ABB RAPID module: Module1.mod

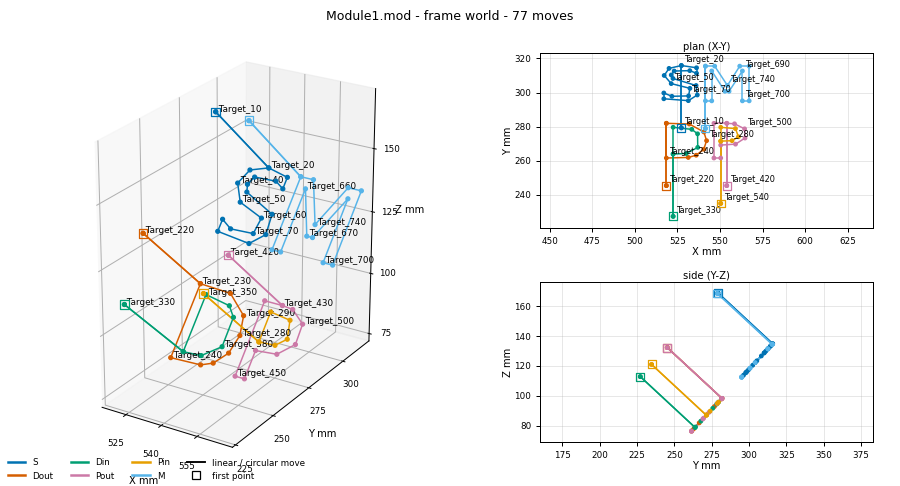
[picture p0: tool path of Module1.mod in frame world, 77 of 79 moves have a stored position in this frame; points joined in program order, loops and branches not executed]
MODULE Module1
        CONST robtarget Target_10:=[[155.704254378,97.181037963,47.999905215],[-0.000000229,0.899659187,0.436592885,-0.000000111],[0,0,-2,0],[9E+09,9E+09,9E+09,9E+09,9E+09,9E+09]];
    CONST robtarget Target_20:=[[155.704254378,97.181063465,-2.000094786],[-0.000000229,0.899659187,0.436592885,-0.000000111],[0,0,-2,0],[9E+09,9E+09,9E+09,9E+09,9E+09,9E+09]];
    CONST robtarget Target_30:=[[162.948986955,99.648648555,-2.000093527],[-0.000000246,0.899659158,0.436592946,0.000000066],[0,0,-2,0],[9E+09,9E+09,9E+09,9E+09,9E+09,9E+09]];
    CONST robtarget Target_40:=[[165.793395383,105.762911115,-2.000090408],[0.00000023,0.899659288,0.436592677,0.000000112],[0,0,-2,0],[9E+09,9E+09,9E+09,9E+09,9E+09,9E+09]];
    CONST robtarget Target_50:=[[161.67264984,112.800998636,-2.000086819],[0.00000023,0.899659288,0.436592677,0.000000111],[0,0,-2,0],[9E+09,9E+09,9E+09,9E+09,9E+09,9E+09]];
    CONST robtarget Target_60:=[[150.659683876,116.873121812,-2.000084742],[0.00000023,0.899659288,0.436592678,0.000000112],[0,0,-2,0],[9E+09,9E+09,9E+09,9E+09,9E+09,9E+09]];
    CONST robtarget Target_70:=[[151.461952919,123.42498567,-2.0000814],[-0.000000248,0.899659158,0.436592944,0.000000058],[0,0,-2,0],[9E+09,9E+09,9E+09,9E+09,9E+09,9E+09]];
    CONST robtarget Target_80:=[[161.259359726,123.777497824,-2.000081221],[-0.00000017,0.899659215,0.436592827,-0.00000019],[0,0,-2,0],[9E+09,9E+09,9E+09,9E+09,9E+09,9E+09]];
    CONST robtarget Target_90:=[[166.012196031,120.908778214,-2.000082684],[-0.000000229,0.899659187,0.436592885,-0.000000111],[0,0,-2,0],[9E+09,9E+09,9E+09,9E+09,9E+09,9E+09]];
    CONST robtarget Target_100:=[[166.012196031,125.916881941,-2.000080129],[0.00000023,0.899659288,0.436592677,0.000000112],[0,0,-2,0],[9E+09,9E+09,9E+09,9E+09,9E+09,9E+09]];
    CONST robtarget Target_110:=[[151.595664427,127.545731212,-2.000079299],[0.00000023,0.899659288,0.436592678,0.000000112],[0,0,-2,0],[9E+09,9E+09,9E+09,9E+09,9E+09,9E+09]];
    CONST robtarget Target_120:=[[146.332293276,122.634872217,-2.000081803],[0.000000229,0.899659287,0.436592678,0.000000111],[0,0,-2,0],[9E+09,9E+09,9E+09,9E+09,9E+09,9E+09]];
    CONST robtarget Target_130:=[[147.049473179,114.454159089,-2.000085976],[-0.000000049,0.899659258,0.436592738,-0.00000025],[0,0,-2,0],[9E+09,9E+09,9E+09,9E+09,9E+09,9E+09]];
    CONST robtarget Target_140:=[[160.627268965,108.376363303,-2.000089076],[-0.00000007,0.899659251,0.436592752,-0.000000245],[0,0,-2,0],[9E+09,9E+09,9E+09,9E+09,9E+09,9E+09]];
    CONST robtarget Target_150:=[[161.636183065,105.349621002,-2.000090619],[0.00000023,0.899659288,0.436592677,0.000000112],[0,0,-2,0],[9E+09,9E+09,9E+09,9E+09,9E+09,9E+09]];
    CONST robtarget Target_160:=[[159.922244653,101.93389977,-2.000092362],[0.00000023,0.899659288,0.436592678,0.000000111],[0,0,-2,0],[9E+09,9E+09,9E+09,9E+09,9E+09,9E+09]];
    CONST robtarget Target_170:=[[150.744773017,101.605698798,-2.000092529],[0.00000023,0.899659288,0.436592678,0.000000111],[0,0,-2,0],[9E+09,9E+09,9E+09,9E+09,9E+09,9E+09]];
    CONST robtarget Target_180:=[[146.782050164,103.890950013,-2.000091364],[0.000000229,0.899659288,0.436592678,0.000000111],[0,0,-2,0],[9E+09,9E+09,9E+09,9E+09,9E+09,9E+09]];
    CONST robtarget Target_190:=[[146.782050164,99.125958117,-2.000093793],[0.00000023,0.899659288,0.436592677,0.000000112],[0,0,-2,0],[9E+09,9E+09,9E+09,9E+09,9E+09,9E+09]];
    CONST robtarget Target_200:=[[155.704254378,97.181063465,-2.000094786],[-0.000000229,0.899659187,0.436592885,-0.000000111],[0,0,-2,0],[9E+09,9E+09,9E+09,9E+09,9E+09,9E+09]];
    CONST robtarget Target_210:=[[155.704254378,97.181037963,47.999905215],[-0.000000229,0.899659187,0.436592885,-0.000000111],[0,0,-2,0],[9E+09,9E+09,9E+09,9E+09,9E+09,9E+09]];
    CONST robtarget Target_220:=[[164.529213859,147.110095762,47.99993068],[0.00000023,0.899659288,0.436592677,0.000000112],[0,0,-2,0],[9E+09,9E+09,9E+09,9E+09,9E+09,9E+09]];
    CONST robtarget Target_230:=[[164.529213859,147.110121263,-2.00006932],[0.00000023,0.899659288,0.436592677,0.000000112],[0,0,-2,0],[9E+09,9E+09,9E+09,9E+09,9E+09,9E+09]];
    CONST robtarget Target_240:=[[164.529213859,177.110121264,-2.00005402],[0.00000023,0.899659288,0.436592677,0.000000112],[0,0,-2,0],[9E+09,9E+09,9E+09,9E+09,9E+09,9E+09]];
    CONST robtarget Target_250:=[[151.632131201,176.6238976,-2.000054268],[0.00000023,0.899659288,0.436592678,0.000000111],[0,0,-2,0],[9E+09,9E+09,9E+09,9E+09,9E+09,9E+09]];
    CONST robtarget Target_260:=[[147.000850812,174.703314133,-2.000055247],[0.000000229,0.899659288,0.436592678,0.000000111],[0,0,-2,0],[9E+09,9E+09,9E+09,9E+09,9E+09,9E+09]];
    CONST robtarget Target_270:=[[142.539748705,169.549343306,-2.000057875],[0.000000228,0.899659287,0.436592679,0.000000112],[0,0,-2,0],[9E+09,9E+09,9E+09,9E+09,9E+09,9E+09]];
    CONST robtarget Target_280:=[[140.87443266,162.134432447,-2.000061658],[0.00000023,0.899659288,0.436592677,0.000000112],[0,0,-2,0],[9E+09,9E+09,9E+09,9E+09,9E+09,9E+09]];
    CONST robtarget Target_290:=[[142.466815156,154.58581008,-2.000065507],[-0.000000003,0.899659272,0.43659271,-0.000000255],[0,0,-2,0],[9E+09,9E+09,9E+09,9E+09,9E+09,9E+09]];
    CONST robtarget Target_300:=[[151.060818397,147.742212025,-2.000068998],[-0.000000194,0.899659205,0.436592848,-0.000000166],[0,0,-2,0],[9E+09,9E+09,9E+09,9E+09,9E+09,9E+09]];
    CONST robtarget Target_310:=[[164.529213859,147.110121263,-2.00006932],[-0.000000229,0.899659187,0.436592885,-0.000000111],[0,0,-2,0],[9E+09,9E+09,9E+09,9E+09,9E+09,9E+09]];
    CONST robtarget Target_320:=[[164.529213859,147.110095762,47.99993068],[-0.000000229,0.899659187,0.436592885,-0.000000111],[0,0,-2,0],[9E+09,9E+09,9E+09,9E+09,9E+09,9E+09]];
    CONST robtarget Target_330:=[[160.542179824,173.657907755,47.999944219],[0.00000023,0.899659288,0.436592677,0.000000112],[0,0,-2,0],[9E+09,9E+09,9E+09,9E+09,9E+09,9E+09]];
    CONST robtarget Target_340:=[[160.542179824,173.657933257,-2.00005578],[0.00000023,0.899659288,0.436592677,0.000000112],[0,0,-2,0],[9E+09,9E+09,9E+09,9E+09,9E+09,9E+09]];
    CONST robtarget Target_350:=[[160.542179824,150.56230927,-2.00006756],[0.00000023,0.899659288,0.436592677,0.000000112],[0,0,-2,0],[9E+09,9E+09,9E+09,9E+09,9E+09,9E+09]];
    CONST robtarget Target_360:=[[149.577836226,152.361336822,-2.000066642],[0.000000229,0.899659287,0.436592678,0.000000112],[0,0,-2,0],[9E+09,9E+09,9E+09,9E+09,9E+09,9E+09]];
    CONST robtarget Target_370:=[[146.174270585,156.190348168,-2.000064689],[0.000000229,0.899659287,0.436592678,0.000000112],[0,0,-2,0],[9E+09,9E+09,9E+09,9E+09,9E+09,9E+09]];
    CONST robtarget Target_380:=[[146.077025853,167.920494035,-2.000058706],[-0.000000195,0.899659159,0.436592943,0.000000163],[0,0,-2,0],[9E+09,9E+09,9E+09,9E+09,9E+09,9E+09]];
    CONST robtarget Target_390:=[[152.847690359,173.232487552,-2.000055997],[-0.000000248,0.899659175,0.43659291,-0.000000061],[0,0,-2,0],[9E+09,9E+09,9E+09,9E+09,9E+09,9E+09]];
    CONST robtarget Target_400:=[[160.542179824,173.657933257,-2.00005578],[-0.000000229,0.899659187,0.436592885,-0.000000111],[0,0,-2,0],[9E+09,9E+09,9E+09,9E+09,9E+09,9E+09]];
    CONST robtarget Target_410:=[[160.542179824,173.657907755,47.999944219],[-0.000000229,0.899659187,0.436592885,-0.000000111],[0,0,-2,0],[9E+09,9E+09,9E+09,9E+09,9E+09,9E+09]];
    CONST robtarget Target_420:=[[129.010575286,147.110095762,47.99993068],[-0.000000229,0.899659187,0.436592885,-0.000000111],[0,0,-2,0],[9E+09,9E+09,9E+09,9E+09,9E+09,9E+09]];
    CONST robtarget Target_430:=[[129.010575286,147.110121263,-2.00006932],[-0.000000229,0.899659187,0.436592885,-0.000000111],[0,0,-2,0],[9E+09,9E+09,9E+09,9E+09,9E+09,9E+09]];
    CONST robtarget Target_440:=[[136.54704206,147.110121263,-2.00006932],[-0.000000229,0.899659187,0.436592885,-0.000000111],[0,0,-2,0],[9E+09,9E+09,9E+09,9E+09,9E+09,9E+09]];
    CONST robtarget Target_450:=[[136.54704206,177.110121264,-2.00005402],[0.00000023,0.899659288,0.436592677,0.000000112],[0,0,-2,0],[9E+09,9E+09,9E+09,9E+09,9E+09,9E+09]];
    CONST robtarget Target_460:=[[132.560008025,177.110121264,-2.00005402],[0.000000229,0.899659288,0.436592678,0.000000111],[0,0,-2,0],[9E+09,9E+09,9E+09,9E+09,9E+09,9E+09]];
    CONST robtarget Target_470:=[[132.560008025,165.926977017,-2.000059724],[0.00000023,0.899659288,0.436592677,0.000000112],[0,0,-2,0],[9E+09,9E+09,9E+09,9E+09,9E+09,9E+09]];
    CONST robtarget Target_480:=[[123.868760051,165.136863565,-2.000060126],[0.000000229,0.899659287,0.436592678,0.000000112],[0,0,-2,0],[9E+09,9E+09,9E+09,9E+09,9E+09,9E+09]];
    CONST robtarget Target_490:=[[118.277187927,159.849181231,-2.000062823],[0.00000023,0.899659287,0.436592678,0.000000112],[0,0,-2,0],[9E+09,9E+09,9E+09,9E+09,9E+09,9E+09]];
    CONST robtarget Target_500:=[[118.53245535,151.887268752,-2.000066884],[-0.00000001,0.89965927,0.436592714,-0.000000254],[0,0,-2,0],[9E+09,9E+09,9E+09,9E+09,9E+09,9E+09]];
    CONST robtarget Target_510:=[[124.464384038,147.54772256,-2.000069097],[-0.000000198,0.899659203,0.436592852,-0.00000016],[0,0,-2,0],[9E+09,9E+09,9E+09,9E+09,9E+09,9E+09]];
    CONST robtarget Target_520:=[[129.010575286,147.110121263,-2.00006932],[-0.000000229,0.899659187,0.436592885,-0.000000111],[0,0,-2,0],[9E+09,9E+09,9E+09,9E+09,9E+09,9E+09]];
    CONST robtarget Target_530:=[[129.010575286,147.110095762,47.99993068],[-0.000000229,0.899659187,0.436592885,-0.000000111],[0,0,-2,0],[9E+09,9E+09,9E+09,9E+09,9E+09,9E+09]];
    CONST robtarget Target_540:=[[132.560008025,162.523385875,47.99993854],[0.00000023,0.899659288,0.436592677,0.000000112],[0,0,-2,0],[9E+09,9E+09,9E+09,9E+09,9E+09,9E+09]];
    CONST robtarget Target_550:=[[132.560008025,162.523411377,-2.00006146],[0.00000023,0.899659288,0.436592677,0.000000112],[0,0,-2,0],[9E+09,9E+09,9E+09,9E+09,9E+09,9E+09]];
    CONST robtarget Target_560:=[[132.560008025,150.56230927,-2.00006756],[0.00000023,0.899659288,0.436592677,0.000000112],[0,0,-2,0],[9E+09,9E+09,9E+09,9E+09,9E+09,9E+09]];
    CONST robtarget Target_570:=[[123.905226825,151.704934878,-2.000066977],[0.000000229,0.899659288,0.436592678,0.000000111],[0,0,-2,0],[9E+09,9E+09,9E+09,9E+09,9E+09,9E+09]];
    CONST robtarget Target_580:=[[122.142666047,158.767333581,-2.000063375],[-0.000000186,0.89965916,0.436592941,0.000000175],[0,0,-2,0],[9E+09,9E+09,9E+09,9E+09,9E+09,9E+09]];
    CONST robtarget Target_590:=[[125.910899435,162.134432447,-2.000061658],[-0.00000025,0.899659173,0.436592914,-0.00000005],[0,0,-2,0],[9E+09,9E+09,9E+09,9E+09,9E+09,9E+09]];
    CONST robtarget Target_600:=[[132.560008025,162.523411377,-2.00006146],[-0.000000229,0.899659187,0.436592885,-0.000000111],[0,0,-2,0],[9E+09,9E+09,9E+09,9E+09,9E+09,9E+09]];
    CONST robtarget Target_610:=[[132.560008025,162.523385875,47.99993854],[-0.000000229,0.899659187,0.436592885,-0.000000111],[0,0,-2,0],[9E+09,9E+09,9E+09,9E+09,9E+09,9E+09]];
    CONST robtarget Target_620:=[[141.555,97.725308454,47.992242797],[0.000000229,0.899659187,0.436592885,-0.000000111],[0,0,-2,0],[9E+09,9E+09,9E+09,9E+09,9E+09,9E+09]];
    CONST robtarget Target_630:=[[141.555,97.715476556,-1.999980632],[0.000000229,0.899659187,0.436592885,-0.000000111],[0,0,-2,0],[9E+09,9E+09,9E+09,9E+09,9E+09,9E+09]];
    CONST robtarget Target_640:=[[141.555,127.716252612,-2.000015929],[0.000000229,0.899659187,0.436592885,-0.000000111],[0,0,-2,0],[9E+09,9E+09,9E+09,9E+09,9E+09,9E+09]];
    CONST robtarget Target_650:=[[137.836,127.716252612,-2.000015929],[0.000000229,0.899659187,0.436592885,-0.000000111],[0,0,-2,0],[9E+09,9E+09,9E+09,9E+09,9E+09,9E+09]];
    CONST robtarget Target_660:=[[137.836,101.87334713,-2.00051431],[0.000000229,0.899659187,0.436592885,-0.000000111],[0,0,-2,0],[9E+09,9E+09,9E+09,9E+09,9E+09,9E+09]];
    CONST robtarget Target_670:=[[130.08,119.450079979,-1.999929472],[0.000000229,0.899659187,0.436592885,-0.000000111],[0,0,-2,0],[9E+09,9E+09,9E+09,9E+09,9E+09,9E+09]];
    CONST robtarget Target_680:=[[127.649,119.450079979,-1.999929472],[0.000000229,0.899659187,0.436592885,-0.000000111],[0,0,-2,0],[9E+09,9E+09,9E+09,9E+09,9E+09,9E+09]];
    CONST robtarget Target_690:=[[119.821,101.87334713,-2.00051431],[0.000000229,0.899659187,0.436592885,-0.000000111],[0,0,-2,0],[9E+09,9E+09,9E+09,9E+09,9E+09,9E+09]];
    CONST robtarget Target_700:=[[119.821,127.716252612,-2.000015929],[0.000000229,0.899659187,0.436592885,-0.000000111],[0,0,-2,0],[9E+09,9E+09,9E+09,9E+09,9E+09,9E+09]];
    CONST robtarget Target_710:=[[115.834,127.716252612,-2.000015929],[0.000000229,0.899659187,0.436592885,-0.000000111],[0,0,-2,0],[9E+09,9E+09,9E+09,9E+09,9E+09,9E+09]];
    CONST robtarget Target_720:=[[115.834,97.715476556,-1.999980632],[0.000000229,0.899659187,0.436592885,-0.000000111],[0,0,-1,0],[9E+09,9E+09,9E+09,9E+09,9E+09,9E+09]];
    CONST robtarget Target_730:=[[121.377,97.715476556,-1.999980632],[0.000000229,0.899659187,0.436592885,-0.000000111],[0,0,-1,0],[9E+09,9E+09,9E+09,9E+09,9E+09,9E+09]];
    CONST robtarget Target_740:=[[128.622,114.417620362,-1.999478829],[0.000000229,0.899659187,0.436592885,-0.000000111],[0,0,-2,0],[9E+09,9E+09,9E+09,9E+09,9E+09,9E+09]];
    CONST robtarget Target_750:=[[136.109,97.715476556,-1.999980632],[0.000000229,0.899659187,0.436592885,-0.000000111],[0,0,-2,0],[9E+09,9E+09,9E+09,9E+09,9E+09,9E+09]];
    CONST robtarget Target_760:=[[141.555,97.715476556,-1.999980632],[0.000000229,0.899659187,0.436592885,-0.000000111],[0,0,-2,0],[9E+09,9E+09,9E+09,9E+09,9E+09,9E+09]];
    CONST robtarget Target_770:=[[141.555,97.725308454,47.992242797],[0.000000229,0.899659187,0.436592885,-0.000000111],[0,0,-2,0],[9E+09,9E+09,9E+09,9E+09,9E+09,9E+09]];
    CONST jointtarget Home:=[[0,0,0,0,0,0],[9E+09,9E+09,9E+09,9E+09,9E+09,9E+09]];
    CONST jointtarget Cerca:=[[0,30,0,0,30,0],[9E+09,9E+09,9E+09,9E+09,9E+09,9E+09]];
!***********************************************************
    !
    ! Module:  Module1
    !
    ! Description:
    !   <Insert description here>
    !
    ! Author: SAMJ
    !
    ! Version: 1.0
    !
    !***********************************************************


    !***********************************************************
    !
    ! Procedure main
    !
    !   This is the entry point of your program
    !
    !***********************************************************
    PROC main()
        GoHome;
        Acercarse;
        S;
        M;
        Din;
        Dout;
        Pin;
        Pout;
        Acercarse;
        GoHome;
    ENDPROC
    PROC S()
        MoveL Target_10,v100,z10,marcador\WObj:=Tablero;
        MoveL Target_20,v100,z10,marcador\WObj:=Tablero;
        MoveL Target_30,v100,z10,marcador\WObj:=Tablero;
        MoveL Target_40,v100,z10,marcador\WObj:=Tablero;
        MoveL Target_50,v100,z10,marcador\WObj:=Tablero;
        MoveL Target_60,v100,z10,marcador\WObj:=Tablero;
        MoveL Target_70,v100,z10,marcador\WObj:=Tablero;
        MoveL Target_80,v100,z10,marcador\WObj:=Tablero;
        MoveL Target_90,v100,z10,marcador\WObj:=Tablero;
        MoveL Target_100,v100,z10,marcador\WObj:=Tablero;
        MoveL Target_110,v100,z10,marcador\WObj:=Tablero;
        MoveL Target_120,v100,z10,marcador\WObj:=Tablero;
        MoveL Target_130,v100,z10,marcador\WObj:=Tablero;
        MoveL Target_140,v100,z10,marcador\WObj:=Tablero;
        MoveL Target_150,v100,z10,marcador\WObj:=Tablero;
        MoveL Target_160,v100,z10,marcador\WObj:=Tablero;
        MoveL Target_170,v100,z10,marcador\WObj:=Tablero;
        MoveL Target_180,v100,z10,marcador\WObj:=Tablero;
        MoveL Target_190,v100,z10,marcador\WObj:=Tablero;
        MoveL Target_200,v100,z10,marcador\WObj:=Tablero;
        MoveL Target_210,v100,z10,marcador\WObj:=Tablero;
    ENDPROC
    PROC Dout()
        MoveL Target_220,v100,z10,marcador\WObj:=Tablero;
        MoveL Target_230,v100,z10,marcador\WObj:=Tablero;
        MoveL Target_240,v100,z10,marcador\WObj:=Tablero;
        MoveL Target_250,v100,z10,marcador\WObj:=Tablero;
        MoveL Target_260,v100,z10,marcador\WObj:=Tablero;
        MoveL Target_270,v100,z10,marcador\WObj:=Tablero;
        MoveL Target_280,v100,z10,marcador\WObj:=Tablero;
        MoveL Target_290,v100,z10,marcador\WObj:=Tablero;
        MoveL Target_300,v100,z10,marcador\WObj:=Tablero;
        MoveL Target_310,v100,z10,marcador\WObj:=Tablero;
        MoveL Target_320,v100,z10,marcador\WObj:=Tablero;
    ENDPROC
    PROC Din()
        MoveL Target_330,v100,z10,marcador\WObj:=Tablero;
        MoveL Target_340,v100,z10,marcador\WObj:=Tablero;
        MoveL Target_350,v100,z10,marcador\WObj:=Tablero;
        MoveL Target_360,v100,z10,marcador\WObj:=Tablero;
        MoveL Target_370,v100,z10,marcador\WObj:=Tablero;
        MoveL Target_380,v100,z10,marcador\WObj:=Tablero;
        MoveL Target_390,v100,z10,marcador\WObj:=Tablero;
        MoveL Target_400,v100,z10,marcador\WObj:=Tablero;
        MoveL Target_410,v100,z10,marcador\WObj:=Tablero;
    ENDPROC
    PROC Pout()
        MoveL Target_420,v100,z10,marcador\WObj:=Tablero;
        MoveL Target_430,v100,z10,marcador\WObj:=Tablero;
        MoveL Target_440,v100,z10,marcador\WObj:=Tablero;
        MoveL Target_450,v100,z10,marcador\WObj:=Tablero;
        MoveL Target_460,v100,z10,marcador\WObj:=Tablero;
        MoveL Target_470,v100,z10,marcador\WObj:=Tablero;
        MoveL Target_480,v100,z10,marcador\WObj:=Tablero;
        MoveL Target_490,v100,z10,marcador\WObj:=Tablero;
        MoveL Target_500,v100,z10,marcador\WObj:=Tablero;
        MoveL Target_510,v100,z10,marcador\WObj:=Tablero;
        MoveL Target_520,v100,z10,marcador\WObj:=Tablero;
        MoveL Target_530,v100,z10,marcador\WObj:=Tablero;
    ENDPROC
    PROC Pin()
        MoveL Target_540,v100,z10,marcador\WObj:=Tablero;
        MoveL Target_550,v100,z10,marcador\WObj:=Tablero;
        MoveL Target_560,v100,z10,marcador\WObj:=Tablero;
        MoveL Target_570,v100,z10,marcador\WObj:=Tablero;
        MoveL Target_580,v100,z10,marcador\WObj:=Tablero;
        MoveL Target_590,v100,z10,marcador\WObj:=Tablero;
        MoveL Target_600,v100,z10,marcador\WObj:=Tablero;
        MoveL Target_610,v100,z10,marcador\WObj:=Tablero;
    ENDPROC
    PROC M()
        MoveL Target_620,v100,z10,marcador\WObj:=Tablero;
        MoveL Target_630,v100,z10,marcador\WObj:=Tablero;
        MoveL Target_640,v100,z10,marcador\WObj:=Tablero;
        MoveL Target_650,v100,z10,marcador\WObj:=Tablero;
        MoveL Target_660,v100,z10,marcador\WObj:=Tablero;
        MoveL Target_670,v100,z10,marcador\WObj:=Tablero;
        MoveL Target_680,v100,z10,marcador\WObj:=Tablero;
        MoveL Target_690,v100,z10,marcador\WObj:=Tablero;
        MoveL Target_700,v100,z10,marcador\WObj:=Tablero;
        MoveL Target_710,v100,z10,marcador\WObj:=Tablero;
        MoveL Target_720,v100,z10,marcador\WObj:=Tablero;
        MoveL Target_730,v100,z10,marcador\WObj:=Tablero;
        MoveL Target_740,v100,z10,marcador\WObj:=Tablero;
        MoveL Target_750,v100,z10,marcador\WObj:=Tablero;
        MoveL Target_760,v100,z10,marcador\WObj:=Tablero;
        MoveL Target_770,v100,z10,marcador\WObj:=Tablero;
    ENDPROC
    PROC GoHome()
        MoveAbsJ Home,v1000,z10,marcador\WObj:=Tablero;
    ENDPROC
    PROC Acercarse()
        MoveAbsJ Cerca,v200,z10,marcador\WObj:=Tablero;
    ENDPROC
ENDMODULE
